FUNCTION_BLOCK FB_LightControl
VAR_IN_OUT
	bTrig1		:	BOOL;
	bTrig2		: 	BOOL;
	bTrig3		: 	BOOL;
END_VAR

{attribute 'TcRpcEnable'}
METHOD Green
bTrig1	:= FALSE;
bTrig2	:= TRUE;
bTrig3	:= FALSE;
END_METHOD

{attribute 'TcRpcEnable'}
METHOD Red
bTrig1	:= TRUE;
bTrig2	:= FALSE;
bTrig3	:= FALSE;
END_METHOD

{attribute 'TcRpcEnable'}
METHOD SwitchOff : BOOL
bTrig1	:= FALSE;
bTrig2	:= FALSE;
bTrig3	:= FALSE;
END_METHOD

{attribute 'TcRpcEnable'}
METHOD White : BOOL
bTrig1	:= FALSE;
bTrig2	:= FALSE;
bTrig3	:= TRUE;
END_METHOD

{attribute 'TcRpcEnable'}
METHOD Yellow : BOOL
bTrig1	:= TRUE;
bTrig2	:= TRUE;
bTrig3	:= FALSE;
END_METHOD

END_FUNCTION_BLOCK

(* stored: Version 1.1.0.1, ProductVersion 3.1.4024.11
   POU FB_LightControl: Id {bc569b6f-d53e-455e-a235-418c41eba51f}, SpecialFunc None
   Method Green: Id {3b537be2-2633-45a3-9ea2-c5a56a734abb}
   Method Red: Id {1f0aa78e-55df-4e06-ba94-b62a7a084276}
   Method SwitchOff: Id {63cbc77a-36fb-4a3c-87c8-b2d1af79befe}
   Method White: Id {2b71246a-d19f-441d-aa2d-cbcd0c06dbaf}
   Method Yellow: Id {ae613c60-aaa8-4916-bf00-efe48abe45c0} *)
